// TIA Portal V18 export
DATA_BLOCK "edelete"   // DB77
VERSION : 0.1
// stored: AutoNumber true, DBAccessibleFromOPCUA true, InstanceOfName Cycle_iterator_spot_generator, InstanceOfType FB
"Cycle_iterator_spot_generator"
   // VAR_INPUT
   //    cur_pos : "typePositions";
   //    "step" : Real;
   //    fullturn : Real := 360.0;
   // END_VAR
   // VAR_OUTPUT
   //    list : "typeSpotList";
   //    ER : Bool;
   // END_VAR
   // VAR
   //    j : Int;
   // END_VAR
BEGIN
END_DATA_BLOCK
